{attribute 'qualified_only'}
VAR_GLOBAL

END_VAR

(* stored: Version 1.1.0.1, ProductVersion 3.1.4024.9
   GVL GVLmqtt: Id {d06ebd27-5bef-4ef1-899c-e2f5b3416f3e} *)
